{attribute 'qualified_only'}
VAR_GLOBAL
	StartButton			: BOOL;
	CarRedLight			: BOOL;
	CarYellowLight		: BOOL;
	CarGreenLight		: BOOL;
	CrossWalkRedLight	: BOOL;
	CrossWalkGreenLight : BOOL;
	NightLight			: BOOL; 
END_VAR

(* stored: Version 1.1.0.1, ProductVersion 3.1.4024.15
   GVL GVL: Id {5881d442-5fa2-4178-8534-e94e56f86ea3} *)
